Omron CX-Programmer project NewProject (CX-Programmer 9.70)

# PLC COKE: CP1L M

## Global symbols (name address type ; comment)
0.00 BOOL  ; Coke
100.00 BOOL  ; Conveyor
100.01 BOOL  ; Robot Arm
100.02 BOOL  ; Taping Cutting
101.00 BOOL  ; LED
1.00 BOOL  ; Start Button
1.01 BOOL  ; Stop
1.02 BOOL  ; reset
T0001 BOOL  ; 3s move
T0002 BOOL  ; 2s Robot Arm
T0003 BOOL  ; 3s move
T0004 BOOL  ; 5s Taping
T0005 BOOL  ; 6s move

## Program NewProgram1 (cyclic task 0)

### Section Section1

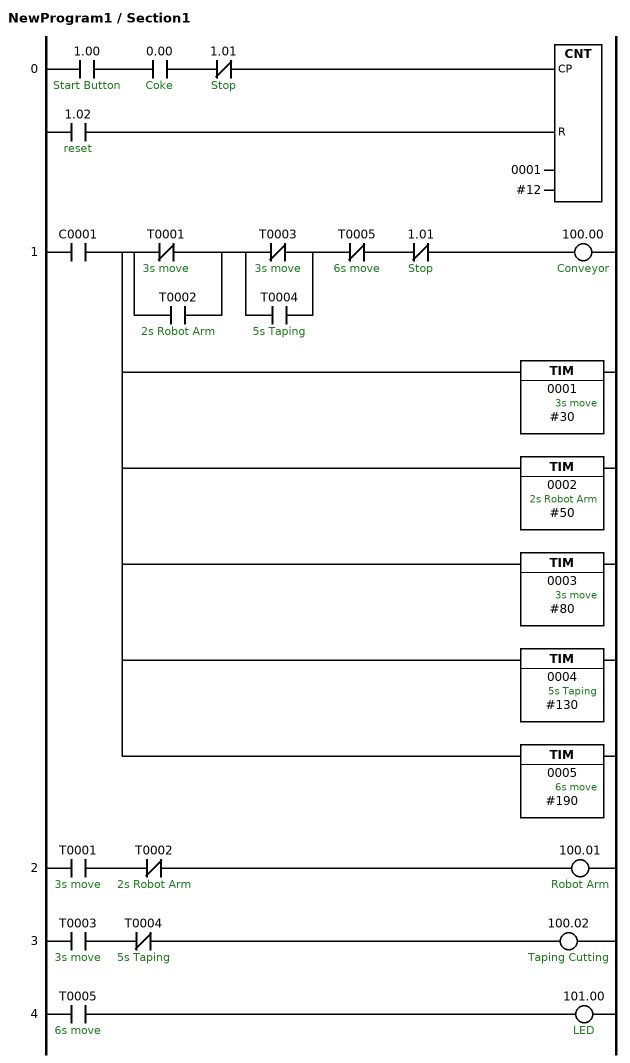
; rung 0
LD 1.00  ; Start Button
AND 0.00  ; Coke
ANDNOT 1.01  ; Stop
LD 1.02  ; reset
CNT 0001 #12
; rung 1
LD C0001
OUT TR0
LDNOT T0001  ; 3s move
OR T0002  ; 2s Robot Arm
ANDLD
LDNOT T0003  ; 3s move
OR T0004  ; 5s Taping
ANDLD
ANDNOT T0005  ; 6s move
ANDNOT 1.01  ; Stop
OUT 100.00  ; Conveyor
LD TR0
TIM 0001 #30  ; 3s move
TIM 0002 #50  ; 2s Robot Arm
TIM 0003 #80  ; 3s move
TIM 0004 #130  ; 5s Taping
TIM 0005 #190  ; 6s move
; rung 2
LD T0001  ; 3s move
ANDNOT T0002  ; 2s Robot Arm
OUT 100.01  ; Robot Arm
; rung 3
LD T0003  ; 3s move
ANDNOT T0004  ; 5s Taping
OUT 100.02  ; Taping Cutting
; rung 4
LD T0005  ; 6s move
OUT 101.00  ; LED

### Section END
; rung 0
END(001)